TYPE EvosensLightConfig EXTENDS DeviceConfiguration :
STRUCT
	SerialCommunication : SerialCommunication;
END_STRUCT
END_TYPE

(* stored: Version 1.1.0.1, ProductVersion 3.1.4024.12
   DUT EvosensLightConfig: Id {9a76cf93-65f7-4b6c-9a6e-a23651c14179} *)
